// TIA Portal project "ERA_Template2Demo" (V15.1)

(* hardware
DEVICE "S71500/ET200MP-Station_1"  S7-1500 station
   slot 0: "Profilschiene_0"  Rack  6ES7 590-1***0-0AA0
   slot 0: "PM 190W 120/230VAC"  PM 190W 120/230VAC  6EP1333-4BA00
   slot 1: "PLC_1"  CPU 1512C-1 PN  6ES7 512-1CK01-0AB0  V2.6
      slot 3: "CPU-Display_1"  6ES7591-1AA00-0AA0
   slot 2: "AQ 4xU/I ST_1"  AQ 4xU/I ST  6ES7 532-5HD00-0AB0  V2.2
*)

// ===== PLC "PLC_1"  CPU 1512C-1 PN =====

VAR_GLOBAL   // PLC tag table "Standard-Variablentabelle"
   "L1" AT %IW0 : Int;   // Füllstand
   "F1" AT %IW2 : Int;   // Durchfluss, regelbare Pumpe
   "P1" AT %IW4 : Int;   // Druck, regelbare Pumpe
   "T1" AT %IW6 : Int;   // Temperatur
   "FC1" AT %QW0 : Int;   // Stellsignal FU für Pumpe M3
   "FC2" AT %QW2 : Int;   // Stellsignal regelbares Ventil
   "B1" AT %I12.0 : Bool;   // Oberer Füllstandsschalter
   "B2" AT %I12.1 : Bool;   // Mittlerer Füllstandsschalter
   "B3" AT %I12.2 : Bool;   // Unterer Füllstandsschalter
   "HS1" AT %I12.3 : Bool;   // Schalter HS1
   "HS2" AT %I12.4 : Bool;   // Schalter HS2
   "HS3" AT %I12.5 : Bool;   // Schalter HS3
   "HS4" AT %I12.6 : Bool;   // Taster HS4
   "HS5" AT %I12.7 : Bool;   // Taster HS5
   "M1" AT %Q6.0 : Bool;   // Pumpe 1, Zulaufpumpe
   "M2" AT %Q6.1 : Bool;   // Pumpe 2, Zulaufpumpe
   "M3" AT %Q6.2 : Bool;   // Pumpe 3, Ablauf
   "M4" AT %Q6.3 : Bool;   // Pumpe 4, Umwälzpumpe
   "LED1" AT %Q6.4 : Bool;   // Lampe 1, Rot
   "LED2" AT %Q6.5 : Bool;   // Lampe 2, Gelb
   "LED3" AT %Q6.6 : Bool;   // Lampe 3, Grün
   "Y1" AT %Q6.7 : Bool;   // Ventil 4
END_VAR

VAR_GLOBAL   // PLC tag table "Pumpanlage"
   "EmergencyStop" AT %I8.0 : Bool;
   "M3_Start" AT %I8.1 : Bool;
   "M1_Start" AT %I8.2 : Bool;
   "M2_Start" AT %I8.3 : Bool;
   "Intial" AT %I8.4 : Bool;
   "Enable" AT %I8.5 : Bool;
   "Enable(1)" AT %I8.6 : Bool;
   "Enable(2)" AT %I8.7 : Bool;
END_VAR

DATA_BLOCK "Programm_DB"   // DB1
{ S7_Optimized_Access := 'TRUE' }
VERSION : 0.1
// stored: InstanceOfName Funktionsbaustein 1
"Funktionsbaustein 1"
BEGIN
END_DATA_BLOCK

DATA_BLOCK "Funktionsbaustein 2_DB"   // DB2
{ S7_Optimized_Access := 'TRUE' }
VERSION : 0.1
// stored: InstanceOfName Funktionsbaustein 2
"Funktionsbaustein 2"
BEGIN
END_DATA_BLOCK

DATA_BLOCK "Funktionsbaustein 3_DB"   // DB3
{ S7_Optimized_Access := 'TRUE' }
VERSION : 0.1
// stored: InstanceOfName Funktionsbaustein 3
"Funktionsbaustein 3"
BEGIN
END_DATA_BLOCK

DATA_BLOCK "Funktionsbaustein 3_DB_1"   // DB4
{ S7_Optimized_Access := 'TRUE' }
VERSION : 0.1
// stored: InstanceOfName Funktionsbaustein 3
"Funktionsbaustein 3"
BEGIN
END_DATA_BLOCK

FUNCTION_BLOCK "Funktionsbaustein 1"   // FB1, FBD
{ S7_Optimized_Access := 'TRUE' }
VERSION : 0.1
BEGIN

REGION Network 1: BEISPIEL
   // Dieses Netzwerk dient nur zur Veranschaulichung. Bitte loeschen bzw. ueberschreiben.
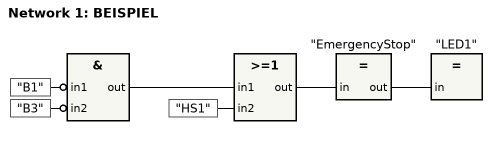
   "EmergencyStop" := (NOT "B1" AND NOT "B3") OR "HS1";
   "LED1" := "EmergencyStop";
END_REGION
END_FUNCTION_BLOCK

FUNCTION_BLOCK "Funktionsbaustein 2"   // FB2, LAD
{ S7_Optimized_Access := 'TRUE' }
VERSION : 0.1
BEGIN

REGION Network 1: Pumpe 3, Ablauf
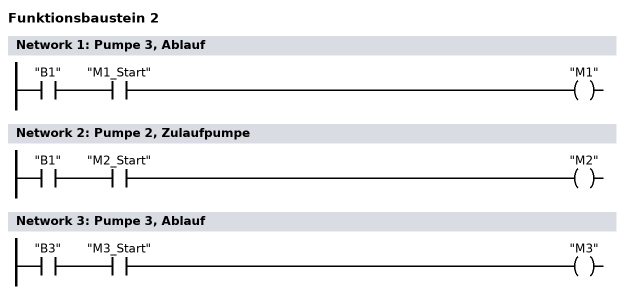
   RUNG wire#powerrail
      Contact( "B1" )
      Contact( "M1_Start" )
      Coil( "M1" )
   END_RUNG
   // the same network as SCL:
   "M1" := "B1" AND "M1_Start";
END_REGION

REGION Network 2: Pumpe 2, Zulaufpumpe
   RUNG wire#powerrail
      Contact( "B1" )
      Contact( "M2_Start" )
      Coil( "M2" )
   END_RUNG
   // the same network as SCL:
   "M2" := "B1" AND "M2_Start";
END_REGION

REGION Network 3: Pumpe 3, Ablauf
   RUNG wire#powerrail
      Contact( "B3" )
      Contact( "M3_Start" )
      Coil( "M3" )
   END_RUNG
   // the same network as SCL:
   "M3" := "B3" AND "M3_Start";
END_REGION
END_FUNCTION_BLOCK

FUNCTION_BLOCK "Funktionsbaustein 3"   // FB3, GRAPH_PLUS
{ S7_Optimized_Access := 'TRUE' }
VERSION : 0.1
   VAR_INPUT
      OFF_SQ : Bool := false;   // Kette ausschalten
      INIT_SQ : Bool := false;   // Kette in Initialzustand versetzen
      ACK_EF : Bool := false;   // Alle Fehler und Störungen quittieren
      S_PREV : Bool := false;   // Vorherigen Schritt am Parameter S_NO ausgeben
      S_NEXT : Bool := false;   // Nächsten Schritt am Parameter S_NO anzeigen
      SW_AUTO : Bool := false;   // Automatischer Betrieb
      SW_TAP : Bool := false;   // Halbautomatisch/Weiterschalten mit Transition
      SW_TOP : Bool := false;   // Halbautomatisch/Ignoriere Transition
      SW_MAN : Bool := false;   // Handbetrieb
      S_SEL : Int := 0;   // Schritt auswählen, der an S_NO ausgegeben werden soll
      S_ON : Bool := false;   // Schritt aktivieren, der an Parameter S_NO anliegt
      S_OFF : Bool := false;   // Schritt deaktivieren, der an Parameter S_NO anliegt
      T_PUSH : Bool := false;   // Schaltfreigabe für Transition im halbautomatischen Betrieb
   END_VAR
   VAR_OUTPUT
      S_NO : Int := 0;   // Schrittnummer
      S_MORE : Bool := false;   // Weitere Schritte sind vorhanden und können in S_NO angezeigt werden.
      S_ACTIVE : Bool := false;   // Schritt, der an Parameter S_NO angezeigt wird, ist aktiv
      ERR_FLT : Bool := false;   // Sammelfehler Interlock oder Supervision
      AUTO_ON : Bool := false;   // Automatischer Betrieb eingeschaltet
      TAP_ON : Bool := false;   // Halbautomatischer Betrieb/Schritt mit Transition eingeschaltet
      TOP_ON : Bool := false;   // Halbautomatischer Betrieb/Ignoriere Transition eingeschaltet
      MAN_ON : Bool := false;   // Handbetrieb eingeschaltet
   END_VAR
   VAR
      enable1 : Bool;
      HMI_INFO : Array[0..8] of UInt;
      IF_PAR : G7_IfParPlus_V6;
      RT_DATA : G7_RTDataPlus_V6;   // Interner Datenbereich
      Trans1 : G7_TransitionPlus_V6;   // Transitionsstruktur
      Trans2 : G7_TransitionPlus_V6;   // Transitionsstruktur
      Trans3 : G7_TransitionPlus_V6;   // Transitionsstruktur
      Trans4 : G7_TransitionPlus_V6;   // Transitionsstruktur
      Trans5 : G7_TransitionPlus_V6;   // Transitionsstruktur
      Trans6 : G7_TransitionPlus_V6;   // Transitionsstruktur
      Trans7 : G7_TransitionPlus_V6;   // Transitionsstruktur
      Trans11 : G7_TransitionPlus_V6;   // Transitionsstruktur
      Trans12 : G7_TransitionPlus_V6;   // Transitionsstruktur
      Trans15 : G7_TransitionPlus_V6;   // Transitionsstruktur
      Step1 : G7_StepPlus_V6;   // Schrittstruktur
      Step2 : G7_StepPlus_V6;   // Schrittstruktur
      Step3 : G7_StepPlus_V6;   // Schrittstruktur
      Step4 : G7_StepPlus_V6;   // Schrittstruktur
      Step5 : G7_StepPlus_V6;   // Schrittstruktur
      Step10 : G7_StepPlus_V6;   // Schrittstruktur
      SINI : Array[0..1] of USInt;
      LSTT : Array[0..9] of USInt;
      ATAJ : Array[0..9] of USInt;
      ATAB : Array[0..9] of USInt;
      PSTT : Array[0..9] of USInt;
      NSTT : Array[0..9] of USInt;
      ASSJ : Array[0..5] of USInt;
      ASSB : Array[0..5] of USInt;
      PTTS : Array[0..5] of USInt;
      NTTS : Array[0..5] of USInt;
      SW_SQTS : Array[0..5] of USInt;
      SWITCH : Array[0..3] of USInt;
      TVX : Array[0..9] of USInt;
      TTX : Array[0..9] of USInt;
      TSX : Array[0..1] of USInt;
      S00X : Array[0..1] of USInt;
      SOFFX : Array[0..1] of USInt;
      SONX : Array[0..1] of USInt;
      SAX : Array[0..1] of USInt;
      SERRX : Array[0..6] of USInt;
      SMX : Array[0..6] of USInt;
      S0X : Array[0..6] of USInt;
      S1X : Array[0..6] of USInt;
      IL_ALARM_INST : Diag_Alarm;
      SUP_ALARM_INST : Diag_Alarm;
      STEP_TIME_ALARM_INST : Diag_Alarm;
      IEC_TIMER_INST : IEC_TIMER;
      TRANSACTION_FLAG : Bool := false;
   END_VAR
   VAR_TEMP
      enabyy : Bool;
      enable : Bool;
   END_VAR
   // SINI[0] := 2;
   // LSTT[0] := 255;
   // LSTT[1] := 255;
   // LSTT[2] := 255;
   // LSTT[3] := 255;
   // LSTT[4] := 255;
   // LSTT[5] := 255;
   // LSTT[6] := 255;
   // LSTT[7] := 255;
   // LSTT[8] := 255;
   // ATAJ[1] := 1;
   // ATAJ[2] := 7;
   // ATAJ[3] := 3;
   // ATAJ[4] := 2;
   // ATAJ[5] := 5;
   // ATAJ[6] := 4;
   // ATAJ[7] := 8;
   // ATAJ[8] := 6;
   // ATAJ[9] := 9;
   // ATAB[1] := 2;
   // ATAB[2] := 1;
   // ATAB[3] := 4;
   // ATAB[4] := 3;
   // ATAB[5] := 6;
   // ATAB[6] := 5;
   // ATAB[7] := 8;
   // ATAB[8] := 7;
   // ATAB[9] := 9;
   // PSTT[1] := 1;
   // PSTT[2] := 1;
   // PSTT[3] := 2;
   // PSTT[4] := 2;
   // PSTT[5] := 3;
   // PSTT[6] := 3;
   // PSTT[7] := 4;
   // PSTT[8] := 4;
   // PSTT[9] := 5;
   // NSTT[0] := 1;
   // NSTT[1] := 2;
   // NSTT[2] := 5;
   // NSTT[3] := 3;
   // NSTT[4] := 5;
   // NSTT[5] := 4;
   // NSTT[6] := 5;
   // NSTT[7] := 5;
   // NSTT[8] := 5;
   // ASSJ[1] := 1;
   // ASSJ[2] := 2;
   // ASSJ[3] := 3;
   // ASSJ[4] := 4;
   // ASSJ[5] := 5;
   // ASSB[1] := 1;
   // ASSB[2] := 2;
   // ASSB[3] := 3;
   // ASSB[4] := 4;
   // ASSB[5] := 5;
   // PTTS[0] := 255;
   // PTTS[2] := 1;
   // PTTS[3] := 3;
   // PTTS[4] := 5;
   // PTTS[5] := 7;
   // NTTS[1] := 1;
   // NTTS[2] := 3;
   // NTTS[3] := 5;
   // NTTS[4] := 7;
   // NTTS[5] := 9;
   // SW_SQTS[2] := 1;
   // SW_SQTS[3] := 2;
   // SW_SQTS[4] := 3;
   // SW_SQTS[5] := 4;
   // TVX[0] := 16#1;
   // TTX[0] := 16#1;
   // TSX[0] := 16#1;
   // S00X[0] := 16#1;
   // SOFFX[0] := 16#1;
   // SONX[0] := 16#1;
   // SAX[0] := 16#1;
   // SERRX[0] := 16#1;
   // SMX[0] := 16#1;
   // S0X[0] := 16#1;
   // S1X[0] := 16#1;
BEGIN
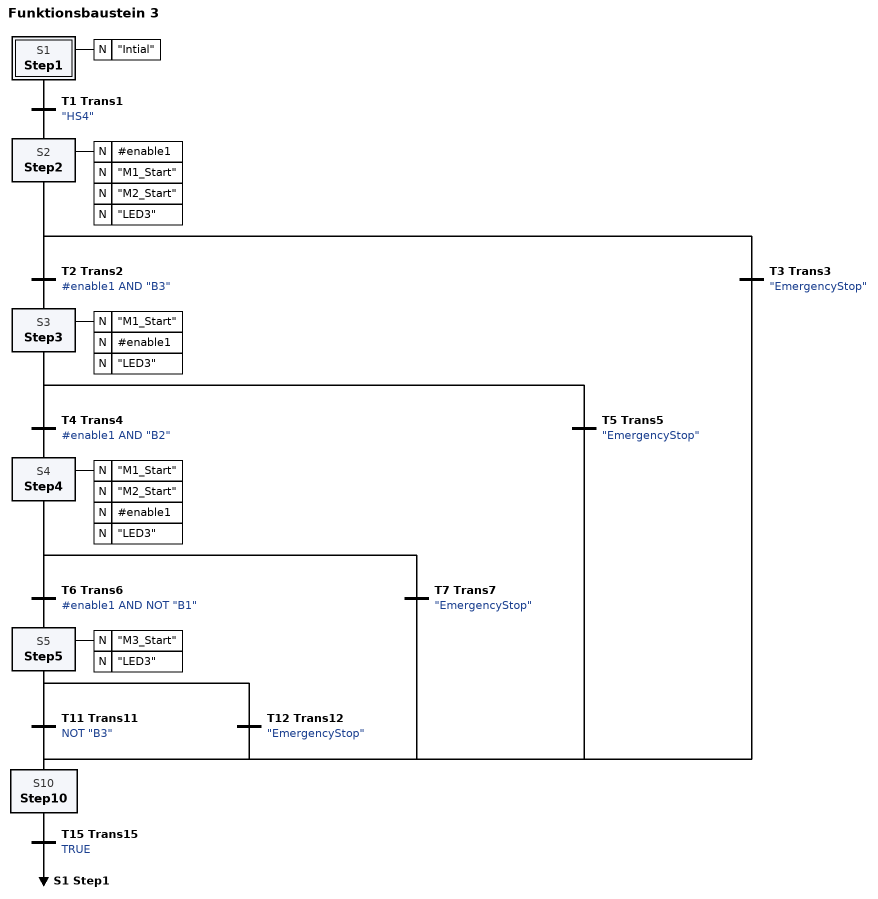
   // sequencer 1
   INITIAL_STEP Step1:   // S1, max time T#10S, warning time T#7S
              N    "Intial"
   END_STEP
   TRANSITION Trans1 FROM Step1 TO Step2   // T1
      := "HS4";
   END_TRANSITION
   STEP Step2:   // S2, max time T#10S, warning time T#7S
              N    #enable1
              N    "M1_Start"
              N    "M2_Start"
              N    "LED3"
   END_STEP
   TRANSITION Trans2 FROM Step2 TO Step3   // T2
      := #enable1 AND "B3";
   END_TRANSITION
   TRANSITION Trans3 FROM Step2 TO Step10   // T3
      := "EmergencyStop";
   END_TRANSITION
   STEP Step3:   // S3, max time T#10S, warning time T#7S
              N    "M1_Start"
              N    #enable1
              N    "LED3"
   END_STEP
   TRANSITION Trans4 FROM Step3 TO Step4   // T4
      := #enable1 AND "B2";
   END_TRANSITION
   TRANSITION Trans5 FROM Step3 TO Step10   // T5
      := "EmergencyStop";
   END_TRANSITION
   STEP Step4:   // S4, max time T#10S, warning time T#7S
              N    "M1_Start"
              N    "M2_Start"
              N    #enable1
              N    "LED3"
   END_STEP
   TRANSITION Trans6 FROM Step4 TO Step5   // T6
      := #enable1 AND NOT "B1";
   END_TRANSITION
   TRANSITION Trans7 FROM Step4 TO Step10   // T7
      := "EmergencyStop";
   END_TRANSITION
   STEP Step5:   // S5, max time T#10S, warning time T#7S
              N    "M3_Start"
              N    "LED3"
   END_STEP
   TRANSITION Trans11 FROM Step5 TO Step10   // T11
      := NOT "B3";
   END_TRANSITION
   TRANSITION Trans12 FROM Step5 TO Step10   // T12
      := "EmergencyStop";
   END_TRANSITION
   STEP Step10:   // S10, max time T#10S, warning time T#7S
   END_STEP
   TRANSITION Trans15 FROM Step10 TO Step1   // T15, jump
      := TRUE;
   END_TRANSITION
END_FUNCTION_BLOCK

ORGANIZATION_BLOCK "Main"   // OB1, LAD, ProgramCycle
TITLE = "Main Program Sweep (Cycle)"
{ S7_Optimized_Access := 'TRUE' }
VERSION : 0.1
   VAR_INPUT
      Initial_Call : Bool;   // Initial call of this OB
      Remanence : Bool;   // =True, if remanent data are available
   END_VAR
   VAR_TEMP   // added for the SCL form of the ladder/FBD networks
      _w1 : Bool;
      _w2 : Bool;
   END_VAR
BEGIN

REGION Network 1
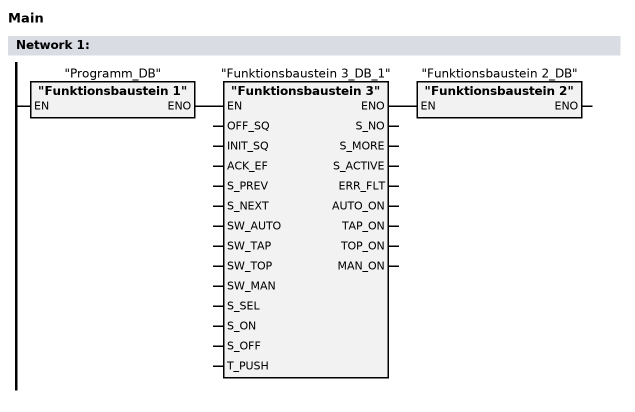
   RUNG wire#powerrail
      "Programm_DB"()
      "Funktionsbaustein 3_DB_1"(OFF_SQ :=, INIT_SQ :=, ACK_EF :=, S_PREV :=, S_NEXT :=, SW_AUTO :=, SW_TAP :=, SW_TOP :=, SW_MAN :=, S_SEL :=, S_ON :=, S_OFF :=, T_PUSH :=, S_NO =>, S_MORE =>, S_ACTIVE =>, ERR_FLT =>, AUTO_ON =>, TAP_ON =>, TOP_ON =>, MAN_ON =>)
      "Funktionsbaustein 2_DB"()
   END_RUNG
   // the same network as SCL:
   "Programm_DB"(ENO => #_w1);   // "Funktionsbaustein 1"
   "Funktionsbaustein 3_DB_1"(EN := #_w1, ENO => #_w2);   // "Funktionsbaustein 3"
   IF #_w2 THEN
       "Funktionsbaustein 2_DB"();   // "Funktionsbaustein 2"
   END_IF;
END_REGION
END_ORGANIZATION_BLOCK